Yaskawa INFORM job: R1_W24(-90,90)KM-OK.JBI

/JOB
//NAME R1_W24(-90,90)KM-OK
///FOLDERNAME KRIS-SCIANA
//POS
///NPOS 57,57,0,5,0,0
///TOOL 0
///POSTYPE PULSE
///PULSE
C00000=123600,-12860,-54312,-41640,88148,80397
C00001=120727,72264,45486,-43419,68187,78537
C00002=120730,72201,41658,-42842,69910,77770
C00003=121913,118625,102550,-47499,60709,82871
C00004=120680,105365,87155,-46138,61919,81546
C00005=120233,105377,87170,-46014,61686,81428
C00006=120680,105365,87155,-46138,61919,81546
C00007=120680,106282,89568,-46525,61204,81923
C00008=120680,105365,87155,-46138,61919,81546
C00009=120680,105137,86855,-46113,61967,81521
C00010=122084,104110,83706,-45998,63689,81381
C00011=120680,105137,86855,-46113,61967,81521
C00012=120282,105147,86868,-46001,61759,81415
C00013=120680,105137,86855,-46113,61967,81521
C00014=120680,105947,89012,-46459,61327,81858
C00015=120680,105137,86855,-46113,61967,81521
C00016=126632,102568,71569,-45370,70765,80217
C00017=105628,110861,70631,9181,76248,77143
C00018=90079,103598,72277,44137,82752,76276
C00019=93115,79989,50120,45682,82697,77911
C00020=94241,81988,53921,45576,81194,77750
C00021=94870,80971,52672,45434,81052,77981
C00022=94241,81988,53921,45576,81194,77750
C00023=94241,82066,55088,45641,80710,77527
C00024=94241,81988,53921,45576,81194,77750
C00025=90439,80786,48344,46103,85116,77771
C00026=91144,88736,58191,46078,83363,77287
C00027=93433,80247,51210,45660,82154,77811
C00028=93989,78186,49515,45558,81861,77938
C00029=94486,77409,48575,45448,81739,78115
C00030=93989,78186,49515,45558,81861,77938
C00031=93989,78219,50499,45608,81441,77746
C00032=93989,78186,49515,45558,81861,77938
C00033=89014,87596,51414,46328,86969,77970
C00034=104117,82222,27161,9419,92014,76171
C00035=117044,66735,15527,-22220,85560,75038
C00036=120735,72113,44062,-43216,68780,78274
C00037=121402,72146,45355,-43635,68530,78708
C00038=124662,56949,12200,-42482,79430,75485
C00039=122936,53754,21123,-42981,73306,77316
C00040=88718,-31891,-11897,-45759,20551,88099
C00041=86773,-38884,-16476,-44684,19033,87459
C00042=94473,-3955,8690,-49143,24744,90031
C00043=97780,-10696,-6647,-43949,30657,87514
C00044=122365,100198,76797,-45341,65431,80657
C00045=120730,72194,45403,-43416,68199,78533
C00046=107638,83716,21915,3272,91251,77584
C00047=122737,105379,80503,39421,63908,84000
C00048=124791,79235,77419,59896,38505,69060
C00049=120735,72112,44061,-43216,68781,78273
C00050=121402,72146,45354,-43635,68530,78708
C00051=124793,78883,76984,59802,38551,69116
C00052=124790,81302,79724,60286,38323,68837
C00053=121233,76069,67571,56949,43092,70676
C00054=123404,106925,84118,39642,62487,83737
C00055=116116,74146,21472,33448,73223,88073
C00056=64895,4412,-70574,32541,79152,65150
BC00000=160885,582527,992696
BC00001=159740,569619,1010808
BC00002=159782,569624,903274
BC00003=165429,568450,884467
BC00004=165429,561459,884467
BC00005=165429,561459,884467
BC00006=165429,561459,884467
BC00007=165429,561459,884467
BC00008=165429,561459,884467
BC00009=148950,487001,914170
BC00010=165429,487001,884467
BC00011=165429,487001,884467
BC00012=165429,487001,884467
BC00013=165429,487001,884467
BC00014=165429,487001,884467
BC00015=165429,487001,884467
BC00016=165429,487001,884467
BC00017=165429,487001,884467
BC00018=165429,462880,884467
BC00019=165429,462880,884467
BC00020=165429,462880,884467
BC00021=165429,462880,884467
BC00022=165429,462880,884467
BC00023=165429,462880,884467
BC00024=165429,462880,884467
BC00025=165429,462880,884467
BC00026=165429,527513,884467
BC00027=165429,527513,884467
BC00028=165429,527513,884467
BC00029=165429,527513,884467
BC00030=165429,527513,884467
BC00031=165429,527513,884467
BC00032=165429,527513,884467
BC00033=165429,527513,884467
BC00034=165777,527440,883097
BC00035=166074,527377,881925
BC00036=167687,568668,876944
BC00037=167687,568668,876944
BC00038=166263,527337,881180
BC00039=166263,527337,881180
BC00040=110119,444193,1058937
BC00041=110177,382782,1058752
BC00042=110177,382782,1058752
BC00043=110177,382782,1058752
BC00044=167434,468990,876574
BC00045=159528,512732,902904
BC00046=167434,540221,876574
BC00047=273098,568941,884467
BC00048=273098,568941,961208
BC00049=167961,630111,877344
BC00050=167961,630111,877344
BC00051=273098,533190,961208
BC00052=273098,474998,961207
BC00053=273098,474998,961207
BC00054=273098,473101,884467
BC00055=273098,515318,884467
BC00056=114596,515318,884467
///POSTYPE BASE
///RECTAN
///RCONF 0,0,0,0,1,0,0,0,0,0,0,0,0,0,0,0,0,0,0,0,0,0,0,0
P00006=2.006,1.622,-0.565,0.0000,0.0000,0.0000
P00021=0.073,2.058,-0.109,0.0000,0.0000,0.0000
P00022=2.006,1.622,-0.565,0.0000,0.0000,0.0000
///RCONF 0,0,0,0,0,0,0,0,0,0,0,0,0,0,0,0,0,0,0,0,0,0,0,0
P00023=-2.957,-4.083,2.762,0.0000,0.0000,0.0000
P00024=-1.466,-0.226,-0.419,0.0000,0.0000,0.0000
//INST
///DATE 2025/04/11 09:46
///ATTR SC,RW
///GROUP1 RB1,BS1
NOP
SFTOF
CALL JOB:CLEAN-R1_LONG
MOVJ C00000 BC00000 VJ=100.00
MOVJ C00001 BC00001 VJ=100.00
MOVJ C00002 BC00002 VJ=100.00
SFTOF
MOVJ C00003 BC00003 VJ=100.00
MOVL C00004 BC00004 V=166.7
REFP 3 C00005 BC00005
CALL JOB:SEARCH-R1
SET P021 P006
SFTON P021
MOVL C00006 BC00006 V=166.7
REFP 3 C00007 BC00007
CALL JOB:SEARCH-R1
SET P021 P006
SFTON P021
MOVL C00008 BC00008 V=166.7
SFTOF
MOVJ C00009 BC00009 VJ=100.00
MOVJ C00010 BC00010 VJ=100.00
MOVL C00011 BC00011 V=166.7
REFP 3 C00012 BC00012
CALL JOB:SEARCH-R1
SET P022 P006
SFTON P022
MOVL C00013 BC00013 V=166.7
REFP 3 C00014 BC00014
CALL JOB:SEARCH-R1
SET P022 P006
SFTON P022
MOVL C00015 BC00015 V=166.7
SFTOF
MOVJ C00016 BC00016 VJ=100.00
MOVJ C00017 BC00017 VJ=30.00
MOVJ C00018 BC00018 VJ=100.00
MOVJ C00019 BC00019 VJ=100.00
MOVL C00020 BC00020 V=166.7
REFP 3 C00021 BC00021
CALL JOB:SEARCH-R1
SET P023 P006
SFTON P023
MOVL C00022 BC00022 V=166.7
REFP 3 C00023 BC00023
CALL JOB:SEARCH-R1
SET P023 P006
SFTON P023
MOVL C00024 BC00024 V=166.7
SFTOF
MOVJ C00025 BC00025 VJ=100.00
MOVJ C00026 BC00026 VJ=100.00
MOVJ C00027 BC00027 VJ=100.00
MOVL C00028 BC00028 V=166.7
REFP 3 C00029 BC00029
CALL JOB:SEARCH-R1
SET P024 P006
SFTON P024
MOVL C00030 BC00030 V=166.7
REFP 3 C00031 BC00031
CALL JOB:SEARCH-R1
SET P024 P006
SFTON P024
MOVL C00032 BC00032 V=166.7
SFTOF
CALL JOB:COFNIJ_DRUT
MOVJ C00033 BC00033 VJ=100.00
MOVJ C00034 BC00034 VJ=30.00
MOVJ C00035 BC00035 VJ=100.00
REFP 1 C00036 BC00036
REFP 2 C00037 BC00037
MOVJ C00038 BC00038 VJ=100.00
SFTON P021
MOVJ C00039 BC00039 VJ=100.00
MOVL C00040 BC00040 V=166.7
MACRO1 MJ#(0) ARGF9
ARCON
SFTON P022
MOVL C00041 BC00041 V=9.2
MOVL C00042 BC00042 V=9.2
ARCOF
SFTOF
MOVL C00043 BC00043 V=666.7
MOVL C00044 BC00044 V=666.7
MOVL C00045 BC00045 V=333.3
MOVJ C00046 BC00046 VJ=100.00
MOVJ C00047 BC00047 VJ=100.00
SFTON P024
MOVL C00048 BC00048 V=166.7 PL=0
REFP 1 C00049 BC00049
REFP 2 C00050 BC00050
MACRO1 MJ#(0) ARGF9
ARCON
MOVL C00051 BC00051 V=9.2
SFTON P023
MOVL C00052 BC00052 V=9.2
ARCOF
SFTOF
MOVL C00053 BC00053 V=666.7
MOVL C00054 BC00054 V=166.7
MOVL C00055 BC00055 V=333.3
MOVJ C00056 BC00056 VJ=100.00
END
